(* Single tank with LimitSwitchLow (piLsLow) and LimitSwitchHigh (piLsHigh)
| using this function when have to DEPENDENT Measure weight
*)
FUNCTION_BLOCK FB_SingleTankV0 EXTENDS FB_SingleTank
VAR
	bAllowInMaterial : BOOL;
	bAllowOutMaterial : BOOL;
	lrWeightWithdraw : LREAL;
END_VAR

bAllowInMaterial := NOT piLsHigh.In;
bAllowOutMaterial := piLslow.In;
SUPER^();

PROPERTY AllowIn : Reference to bool
GET
AllowIn ref= bAllowInMaterial;
END_GET
END_PROPERTY

(*
| Check the minimum condition  (lrWeight > lrLimitMinWeight
								AND piLslow.In;)
*)
PROPERTY AllowOut : REFERENCE TO BOOL
GET
AllowOut ref= bAllowOutMaterial;
END_GET
END_PROPERTY

PROPERTY WeightWithdraw : lreal
GET
WeightWithdraw := lrWeightWithdraw;
END_GET
SET
lrWeightWithdraw := WeightWithdraw;
END_SET
END_PROPERTY

END_FUNCTION_BLOCK

(* stored: Version 1.1.0.1, ProductVersion 3.1.4024.12
   POU FB_SingleTankV0: Id {804ff059-bff6-46a3-be72-e0e118682176}, SpecialFunc None
   Property AllowIn: Id {fc712f05-a064-4a5a-96e7-72aaec14e8cf}
   Get Get: Id {5c729add-9dbd-4aa3-b258-be82a8761357}
   Property AllowOut: Id {0e0965dc-bf3f-4465-bfeb-792393b01443}
   Get Get: Id {b01519fc-927a-40ec-ba86-a2b2d4e2c6ab}
   Property WeightWithdraw: Id {29fd68ca-7307-4b79-a062-bfa4580def3d}
   Get Get: Id {f4d324d7-bfd5-43b4-ba04-e024cc8f3469}
   Set Set: Id {c577a9a8-e76c-427f-bdd9-14600dcf32e2} *)
